FUNCTION F_LminToEng : LREAL
VAR_INPUT
	fLminFlow : LREAL;
END_VAR
VAR
END_VAR

F_LminToEng := fLminFlow / 60000;

END_FUNCTION

(* stored: Version 1.1.0.1, ProductVersion 3.1.4024.10
   POU F_LminToEng: Id {575677ff-2a4b-4d5e-af39-dad63e3f7450}, SpecialFunc None *)
